TYPE Mat3d : ARRAY[1..3, 1..3] OF LREAL; END_TYPE

(* stored: Version 1.1.0.1, ProductVersion 3.1.4024.12
   DUT Mat3d: Id {3a1d61ee-65b6-4522-a2a2-1332e03f6011} *)
